FUNCTION_BLOCK FieldsToArrowheadSystem (* Translate individual fields to an ArrowheadSystem type *)
  (* Standard: 61499-2; Description: Copyright (c) 2018 fortiss GmbH This program and the accompanying materials are made available under the terms of the Eclipse Public License 2.0 which is available at https://www.eclipse.org/legal/epl-2.0/ SPDX-License-Identifier: EPL-2.0 *)
  (* Version 1.0, 2018-09-21, Jose Cabral, fortiss GmbH *)
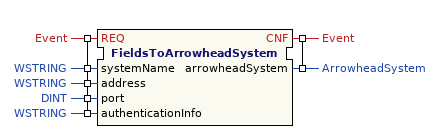
  EVENT_INPUT
    REQ WITH authenticationInfo, port, address, systemName; (* Create arrowhead system *)
  END_EVENT
  EVENT_OUTPUT
    CNF WITH arrowheadSystem; (* Arrowhead system created *)
  END_EVENT
  VAR_INPUT
    systemName : WSTRING; (* Identification of the system *)
    address : WSTRING; (* Address of the offered services *)
    port : DINT; (* Port of the of the offered services *)
    authenticationInfo : WSTRING; (* Authentication info of the system *)
  END_VAR
  VAR_OUTPUT
    arrowheadSystem : ArrowheadSystem; (* Created Arrowhead system *)
  END_VAR
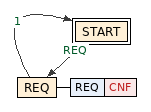
  EC_STATES
    START; (* Initial State *)
    REQ : REQ -> CNF; (* Normal execution *)
  END_STATES
  EC_TRANSITIONS
    START TO REQ := REQ;
    REQ TO START := 1;
  END_TRANSITIONS
  ALGORITHM REQ IN ST: (* Normally executed algorithm *)
arrowheadSystem.systemName := systemName;
arrowheadSystem.address := address;
arrowheadSystem.port := port;
arrowheadSystem.authenticationInfo := authenticationInfo;
  END_ALGORITHM
END_FUNCTION_BLOCK
